{attribute 'qualified_only'}
{attribute 'strict'}
TYPE TunePhase :
(
	init,
	baseline,
	step,
	processData,
	done
);
END_TYPE

(* stored: Version 1.1.0.1, ProductVersion 3.1.4024.12
   DUT TunePhase: Id {50fd9f01-84de-437e-9a07-0c552a3bed8c} *)
